(* IEC 61131-3 sources: 89152_FlorisHendrix_AfstudeerProject/89152_FlorisHendrix_ExamenProject/Stations/Terminal/HMI/Class/_ToolCat, 1 file *)

(* ---- _ToolCat.st ---- *)
(*!
<Class
	Name               = "_ToolCat"
	Revision           = "1.1"
	RealtimeTask       = "false"
	CyclicTask         = "false"
	BackgroundTask     = "false"
	Sigmatek           = "true"
	OSInterface        = "false"
	HighPriority       = "false"
	Automatic          = "false"
	UpdateMode         = "Prescan"
	SharedCommandTable = "true"
	Objectsize         = "(284,120)"
	Comment            = "load and save machinedata to any physical device">
	<Channels>
		<Server Name="Server0" Visualized="true" Initialize="false" WriteProtected="true" Retentive="false"/>
		<Client Name="Lse" Required="true" Internal="false"/>
	</Channels>
	<RevDoku>
		<Owner/>
		<Dokumentation Revision="1.1" Date="2019-04-23" Author="kolott" Company="sigmatek" Description="sa42046: new virtual method LoadLabelEx() added"/>
		<Dokumentation Revision="1.0" Date="2017-07-13" Author="kolott" Company="sigmatek" Description="sa37331: 2 new methods (LoadLabel() and SaveLabel())"/>
	</RevDoku>
</Class>
*)
_ToolCat : CLASS
  //Servers:
	Server0 	: SvrChCmd_DINT;
  //Clients:
	Lse 	: CltChCmd__Lse;
  //Variables:
  //Functions:

	FUNCTION VIRTUAL GLOBAL Init;

	FUNCTION __CDECL VIRTUAL GLOBAL LoadStart
		VAR_INPUT
			pdata 	: ^_TOOLDATA;
		END_VAR
		VAR_OUTPUT
			retcode (AL) 	: BOOL;
		END_VAR;

	FUNCTION __CDECL VIRTUAL GLOBAL LoadRun
		VAR_INPUT
			pdata 	: ^_TOOLDATA;
			pres 	: ^_RESULT;
			pvar 	: ^_VARIABLE;
			pvl 	: ^_VARLABEL;
		END_VAR
		VAR_OUTPUT
			retcode (AL) 	: BOOL;
		END_VAR;

	FUNCTION __CDECL VIRTUAL GLOBAL LoadEnd
		VAR_INPUT
			pdata 	: ^_TOOLDATA;
		END_VAR;

	FUNCTION __CDECL VIRTUAL GLOBAL SaveStart
		VAR_INPUT
			pdata 	: ^_TOOLDATA;
		END_VAR
		VAR_OUTPUT
			retcode (AL) 	: BOOL;
		END_VAR;

	FUNCTION __CDECL VIRTUAL GLOBAL SaveRun
		VAR_INPUT
			pdata 	: ^_TOOLDATA;
			label 	: ^_ASCII;
			pvl 	: ^_VARIABLE;
		END_VAR
		VAR_OUTPUT
			retcode (AL) 	: BOOL;
		END_VAR;

	FUNCTION __CDECL VIRTUAL GLOBAL SaveEnd
		VAR_INPUT
			pdata 	: ^_TOOLDATA;
		END_VAR;

	FUNCTION __CDECL VIRTUAL GLOBAL ErrorOccured
		VAR_INPUT
			pdata 	: ^_TOOLDATA;
			pres 	: ^_RESULT;
			pvar 	: ^_VARIABLE;
			pvl 	: ^_VARLABEL;
		END_VAR
		VAR_OUTPUT
			retcode (AL) 	: BOOL;
		END_VAR;

	FUNCTION __CDECL VIRTUAL GLOBAL IdleRun
		VAR_INPUT
			pdata 	: ^_TOOLDATA;
		END_VAR
		VAR_OUTPUT
			retcode (AL) 	: BOOL;
		END_VAR;
				//! <Function Comment="method will be called right before variable will be written to file.&#13;&#10;pdata... pointer to tooldata&#13;&#10;label ... pointer to variablelabel&#13;&#10;station ... stationnumber of variable to write&#13;&#10;return &apos;true&apos; when variable should be written in file, on the other hand &apos;false&apos;." Name="SaveLabel"/>
	FUNCTION __CDECL VIRTUAL GLOBAL SaveLabel
		VAR_INPUT
			pdata 	: ^_TOOLDATA;
			label 	: ^CHAR;
			station 	: UDINT;
		END_VAR
		VAR_OUTPUT
			retcode (AL) 	: BOOL;
		END_VAR;
				//! <Function Comment="method will be called right before variable will be stored into machine.&#13;&#10;pdate... pointer to tooldata&#13;&#10;label ... pointer to variablelabel&#13;&#10;station ... stationnumber of variable to store&#13;&#10;return &apos;true&apos; when variable should be stored into machine, on the other hand &apos;false&apos;." Name="LoadLabel"/>
	FUNCTION __CDECL VIRTUAL GLOBAL LoadLabel
		VAR_INPUT
			pdata 	: ^_TOOLDATA;
			label 	: ^CHAR;
			station 	: UDINT;
		END_VAR
		VAR_OUTPUT
			retcode (AL) 	: BOOL;
		END_VAR;
				//! <Function Comment="method will be called right before variable will be stored into machine.&#13;&#10;pdate... pointer to tooldata&#13;&#10;label ... pointer to variablelabel&#13;&#10;pstation ... pointer to stationnumber of variable to store&#13;&#10;return &apos;true&apos; when variable should be stored into machine, on the other hand &apos;false&apos;." Name="LoadLabelEx"/>
	FUNCTION __CDECL VIRTUAL GLOBAL LoadLabelEx
		VAR_INPUT
			pdata 	: ^_TOOLDATA;
			label 	: ^CHAR;
			pstation 	: ^UDINT;
		END_VAR
		VAR_OUTPUT
			retcode (AL) 	: BOOL;
		END_VAR;
  //Tables:
	FUNCTION @STD
		VAR_OUTPUT
			ret_code	: CONFSTATES;
		END_VAR;
	FUNCTION GLOBAL TAB @CT_;
END_CLASS;

#pragma usingLtd _Lse

//*********************Inserted from .\_ToolCat\_ToolCat_00_00.st*********************

#pragma warning (disable: 73)

FUNCTION VIRTUAL GLOBAL _ToolCat::Init

  if(_firstscan) then
    if(IsClientConnected(#Lse)) then
      Lse.SetThisPointer(this$^void, 0);
    end_if;
  end_if;

END_FUNCTION
FUNCTION __CDECL VIRTUAL GLOBAL _ToolCat::LoadStart
VAR_INPUT
	pdata   : ^_TOOLDATA;
END_VAR
VAR_OUTPUT
	retcode		: BOOL;
END_VAR

  retcode := TRUE;

//  pdata^.care_state := pdata^.care_state or NOCARE_LIMITS;

END_FUNCTION
FUNCTION __CDECL VIRTUAL GLOBAL _ToolCat::LoadRun
VAR_INPUT
	pdata : ^_TOOLDATA;
	pres  : ^_RESULT;
	pvar  : ^_VARIABLE;
	pvl   : ^_VARLABEL;
END_VAR
VAR_OUTPUT
	retcode		: BOOL;
END_VAR

  retcode := TRUE;

END_FUNCTION
FUNCTION __CDECL VIRTUAL GLOBAL _ToolCat::LoadEnd
VAR_INPUT
	pdata   : ^_TOOLDATA;
END_VAR

END_FUNCTION
FUNCTION __CDECL VIRTUAL GLOBAL _ToolCat::SaveStart
VAR_INPUT
	pdata   : ^_TOOLDATA;
END_VAR
VAR_OUTPUT
	retcode		: BOOL;
END_VAR

  retcode := TRUE;

END_FUNCTION
FUNCTION __CDECL VIRTUAL GLOBAL _ToolCat::SaveRun
VAR_INPUT
	pdata   : ^_TOOLDATA;
	label	: ^_ASCII;
	pvl		: ^_VARIABLE;
END_VAR
VAR_OUTPUT
	retcode		: BOOL;
END_VAR

  retcode := TRUE;

END_FUNCTION
FUNCTION __CDECL VIRTUAL GLOBAL _ToolCat::SaveEnd
VAR_INPUT
	pdata   : ^_TOOLDATA;
END_VAR

END_FUNCTION
FUNCTION __CDECL VIRTUAL GLOBAL _ToolCat::ErrorOccured
VAR_INPUT
	pdata : ^_TOOLDATA;
	pres  : ^_RESULT;
	pvar  : ^_VARIABLE;
	pvl   : ^_VARLABEL;
END_VAR
VAR_OUTPUT
	retcode		: BOOL;
END_VAR

  // retcode := TRUE  system should go on like nothing happend
  // retcode := FALSE remain in error state

  retcode := true;

  case(pdata^.ToolError) of
    TE_CANTOPEN      ,
    TE_NO_TOOLCAT    ,
    TE_DISK_ERROR    ,
    TE_TOOLESSMEMORY ,
    TE_INVALID_CRC   : retcode := false;
//    TE_CANTSAVEENTRY
//    TE_NO_STATESCHEME,           // ungültiges statescheme
//    TE_NO_ACCESS,                // kein access
//    TE_NO_CHKBIT,                // ungültiges chkbit
//    TE_ERROR_LIMITS,             // grenzwertverletzung
//    TE_UNKNOWN_SERVER,           // unbekannter server
//    TE_UNKNOWN_LINE_FORMAT,      // unbekannter fileeintrag
//    TE_FILTER_DOESNT_FIT,        // filter passt nicht
  end_case;

END_FUNCTION

FUNCTION __CDECL VIRTUAL GLOBAL _ToolCat::IdleRun
VAR_INPUT
	pdata		: ^_TOOLDATA;
END_VAR
VAR_OUTPUT
	retcode		: bool;
END_VAR

  retcode := true;

END_FUNCTION //__CDECL VIRTUAL GLOBAL _ToolCat::IdleRun

FUNCTION __CDECL VIRTUAL GLOBAL _ToolCat::SaveLabel
	VAR_INPUT
		pdata 	: ^_TOOLDATA;
		label 	: ^CHAR;
		station 	: UDINT;
	END_VAR
	VAR_OUTPUT
		retcode 	: BOOL;
	END_VAR

  retcode := true;

END_FUNCTION

FUNCTION __CDECL VIRTUAL GLOBAL _ToolCat::LoadLabel
	VAR_INPUT
		pdata 	: ^_TOOLDATA;
		label 	: ^CHAR;
		station 	: UDINT;
	END_VAR
	VAR_OUTPUT
		retcode 	: BOOL;
	END_VAR

  retcode := true;

END_FUNCTION

FUNCTION __CDECL VIRTUAL GLOBAL _ToolCat::LoadLabelEx
	VAR_INPUT
		pdata 	: ^_TOOLDATA;
		label 	: ^CHAR;
		pstation 	: ^UDINT;
	END_VAR
	VAR_OUTPUT
		retcode 	: BOOL;
	END_VAR

  retcode := true;

END_FUNCTION
